{attribute 'conditionalshow'}
FUNCTION_BLOCK FB_CV_ULINT_TO_WORD
VAR_INPUT
	{attribute 'hide'}
	uliInputValue				: ULINT;							//Input value that is converted into the output value			
	{attribute 'hide'}				
	eByteOrderForConvert		: eByteOrder;						//Byte Format
END_VAR
VAR_OUTPUT
	{attribute 'hide'}
	wOutputValue_1				: WORD;								//Converted output value
	{attribute 'hide'}
	wOutputValue_2				: WORD;								//Converted output value
	{attribute 'hide'}
	wOutputValue_3				: WORD;								//Converted output value
	{attribute 'hide'}
	wOutputValue_4				: WORD;								//Converted output value
END_VAR
VAR
END_VAR

//Creator : Kai Ebensperger
//Company : Lynus AG
//Date : 28.04.2021
//Version : 1.0.0.0

//With this functionblock its possible to convert a certain Datatyp in a other Datatype
//The byte order can be selected between BigEndian and LittleEndian
//ULINT TO WORD
//Created for the Edge Device Lib over Modbus TCP
//Modbus TCP is WORD oriented

IF eByteOrderForConvert = eByteOrder.eBigEndian THEN
	wOutputValue_1 := ULINT_TO_WORD(SHR(uliInputValue,48) AND 16#FFFF);
	wOutputValue_2 := ULINT_TO_WORD(SHR(uliInputValue,32) AND 16#FFFF);
	wOutputValue_3 := ULINT_TO_WORD(SHR(uliInputValue,16) AND 16#FFFF);
	wOutputValue_4 := ULINT_TO_WORD(uliInputValue) AND 16#FFFF;
ELSE
	wOutputValue_4 := ULINT_TO_WORD(SHR(uliInputValue,48) AND 16#FFFF);
	wOutputValue_3 := ULINT_TO_WORD(SHR(uliInputValue,32) AND 16#FFFF);
	wOutputValue_2 := ULINT_TO_WORD(SHR(uliInputValue,16) AND 16#FFFF);
	wOutputValue_1 := ULINT_TO_WORD(uliInputValue) AND 16#FFFF;
END_IF

END_FUNCTION_BLOCK

(* stored: Version 1.1.0.1, ProductVersion 3.1.4024.9
   POU FB_CV_ULINT_TO_WORD: Id {1b2a9c33-0e93-4e9f-8c65-026614c57728}, SpecialFunc None *)
